INTERFACE I_FileSystemEntryCollection EXTENDS __SYSTEM.IQueryInterface, I_Collection

METHOD Clear
END_METHOD

METHOD GetFirst : I_FileSystemEntry
END_METHOD

METHOD GetNext : I_FileSystemEntry
VAR_INPUT
	Entry : I_FileSystemEntry;
END_VAR
END_METHOD

METHOD Insert
VAR_INPUT
	Entry : I_FileSystemEntry;
END_VAR
END_METHOD

END_INTERFACE

(* stored: Version 1.1.0.1, ProductVersion 3.1.4024.9
   Itf I_FileSystemEntryCollection: Id {2eefa4f4-b620-4403-9654-87d5923b0013}
   Method Clear: Id {ba765080-6bd7-4248-81cd-65eba6d697a4}
   Method GetFirst: Id {5d1ec355-1838-4d2c-a8c0-71a7c4a8d413}
   Method GetNext: Id {4e41c67e-821b-454d-8be3-531df4a11fef}
   Method Insert: Id {56e0fe63-4afd-45e7-b9f2-cf80ab8f1e1b} *)
